// TIA Portal V20 export
FUNCTION_BLOCK "FB_MABS_PNIO"   // FB6, LAD
// stored: Access Published, MemoryReserve 100, Namespace Global, SetENOAutomatically false
   VAR_IN_OUT
      IBP_in : "IB_P01/02/03_in_64bytes_struct";
      IBP_out : "IB_P01/02/03_out_64bytes_struct";
      MABS : "Global.MABS";
   END_VAR
   VAR
      Initializing : Bool;
      Waiting_sw_req : Bool;
      Switching_left : Bool;
      "Switching_left to straight" : Bool;
      "Switching_right to straight" : Bool;
      Switching_right : Bool;
      Switching_done : Bool;
      Tof_life_bit { S7_SetPoint := 'True'} : TON_TIME;
      MABS_sw_timout { S7_SetPoint := 'True'} : TON_TIME;
      "position status_right" : Bool;
      "position status_left" : Bool;
      "position status_straight" : Bool;
      Edge0 : Bool;
      Edge1 : Bool;
      Edge2 : Bool;
      Edge3 : Bool;
      Edge4 : Bool;
      Edge5 : Bool;
      Edge6 : Bool;
      Ton_err_motor_A { S7_SetPoint := 'True'} : TON_TIME;
      Ton_err_motor_B { S7_SetPoint := 'True'} : TON_TIME;
      Ton_err_motor_Com { S7_SetPoint := 'True'} : TON_TIME;
   END_VAR
   VAR_TEMP
      Temp_err_com : Bool;
   END_VAR
   VAR_TEMP   // added for the SCL form of the ladder/FBD networks
      _w1 : Bool;
      _w2 : Bool;
   END_VAR
BEGIN

REGION Network 1: Error motor A & B
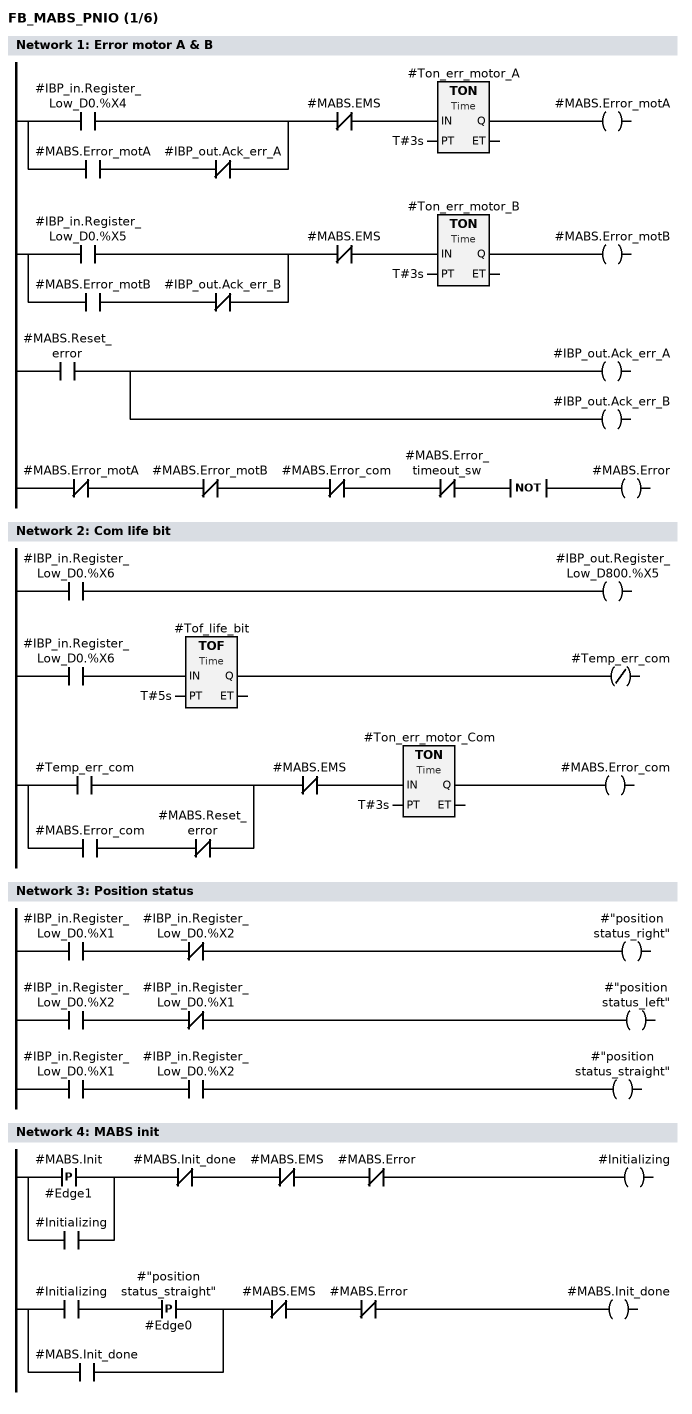
   RUNG wire#powerrail
      Contact( #IBP_in.Register_Low_D0.%X4 )
      wire#w1
      I_Contact( #MABS.EMS )
      { S7_Templates := "time_type := Time" } #Ton_err_motor_A.TON(pt := T#3s, et =>)
      Coil( #MABS.Error_motA )
   END_RUNG
   RUNG wire#powerrail
      Contact( #MABS.Error_motA )
      I_Contact( #IBP_out.Ack_err_A )
   END_RUNG wire#w1
   RUNG wire#powerrail
      Contact( #IBP_in.Register_Low_D0.%X5 )
      wire#w2
      I_Contact( #MABS.EMS )
      { S7_Templates := "time_type := Time" } #Ton_err_motor_B.TON(pt := T#3s, et =>)
      Coil( #MABS.Error_motB )
   END_RUNG
   RUNG wire#powerrail
      Contact( #MABS.Error_motB )
      I_Contact( #IBP_out.Ack_err_B )
   END_RUNG wire#w2
   RUNG wire#powerrail
      Contact( #MABS.Reset_error )
      wire#w3
      Coil( #IBP_out.Ack_err_A )
   END_RUNG
   RUNG wire#w3
      Coil( #IBP_out.Ack_err_B )
   END_RUNG
   RUNG wire#powerrail
      I_Contact( #MABS.Error_motA )
      I_Contact( #MABS.Error_motB )
      I_Contact( #MABS.Error_com )
      I_Contact( #MABS.Error_timeout_sw )
      Not()
      Coil( #MABS.Error )
   END_RUNG
   // the same network as SCL:
   #Ton_err_motor_A(IN := (#IBP_in.Register_Low_D0.%X4 OR (#MABS.Error_motA AND NOT #IBP_out.Ack_err_A)) AND NOT #MABS.EMS,   // TON
                    PT := T#3s);
   #MABS.Error_motA := #Ton_err_motor_A.Q;
   #Ton_err_motor_B(IN := (#IBP_in.Register_Low_D0.%X5 OR (#MABS.Error_motB AND NOT #IBP_out.Ack_err_B)) AND NOT #MABS.EMS,   // TON
                    PT := T#3s);
   #MABS.Error_motB := #Ton_err_motor_B.Q;
   #IBP_out.Ack_err_A := #MABS.Reset_error;
   #IBP_out.Ack_err_B := #MABS.Reset_error;
   #MABS.Error := NOT (NOT #MABS.Error_motA AND NOT #MABS.Error_motB AND NOT #MABS.Error_com AND NOT #MABS.Error_timeout_sw);
END_REGION

REGION Network 2: Com life bit
   RUNG wire#powerrail
      Contact( #IBP_in.Register_Low_D0.%X6 )
      Coil( #IBP_out.Register_Low_D800.%X5 )
   END_RUNG
   RUNG wire#powerrail
      Contact( #IBP_in.Register_Low_D0.%X6 )
      { S7_Templates := "time_type := Time" } #Tof_life_bit.TOF(pt := T#5s, et =>)
      I_Coil( #Temp_err_com )
   END_RUNG
   RUNG wire#powerrail
      Contact( #Temp_err_com )
      wire#w1
      I_Contact( #MABS.EMS )
      { S7_Templates := "time_type := Time" } #Ton_err_motor_Com.TON(pt := T#3s, et =>)
      Coil( #MABS.Error_com )
   END_RUNG
   RUNG wire#powerrail
      Contact( #MABS.Error_com )
      I_Contact( #MABS.Reset_error )
   END_RUNG wire#w1
   // the same network as SCL:
   #IBP_out.Register_Low_D800.%X5 := #IBP_in.Register_Low_D0.%X6;
   #Tof_life_bit(IN := #IBP_in.Register_Low_D0.%X6, PT := T#5s);   // TOF
   #Temp_err_com := NOT #Tof_life_bit.Q;
   #Ton_err_motor_Com(IN := (#Temp_err_com OR (#MABS.Error_com AND NOT #MABS.Reset_error)) AND NOT #MABS.EMS,   // TON
                      PT := T#3s);
   #MABS.Error_com := #Ton_err_motor_Com.Q;
END_REGION

REGION Network 3: Position status
   RUNG wire#powerrail
      Contact( #IBP_in.Register_Low_D0.%X1 )
      I_Contact( #IBP_in.Register_Low_D0.%X2 )
      Coil( #"position status_right" )
   END_RUNG
   RUNG wire#powerrail
      Contact( #IBP_in.Register_Low_D0.%X2 )
      I_Contact( #IBP_in.Register_Low_D0.%X1 )
      Coil( #"position status_left" )
   END_RUNG
   RUNG wire#powerrail
      Contact( #IBP_in.Register_Low_D0.%X1 )
      Contact( #IBP_in.Register_Low_D0.%X2 )
      Coil( #"position status_straight" )
   END_RUNG
   // the same network as SCL:
   #"position status_right" := #IBP_in.Register_Low_D0.%X1 AND NOT #IBP_in.Register_Low_D0.%X2;
   #"position status_left" := #IBP_in.Register_Low_D0.%X2 AND NOT #IBP_in.Register_Low_D0.%X1;
   #"position status_straight" := #IBP_in.Register_Low_D0.%X1 AND #IBP_in.Register_Low_D0.%X2;
END_REGION

REGION Network 4: MABS init
   RUNG wire#powerrail
      P_Contact(operand := #MABS.Init, bit := #Edge1)
      wire#w1
      I_Contact( #MABS.Init_done )
      I_Contact( #MABS.EMS )
      I_Contact( #MABS.Error )
      Coil( #Initializing )
   END_RUNG
   RUNG wire#powerrail
      Contact( #Initializing )
   END_RUNG wire#w1
   RUNG wire#powerrail
      Contact( #Initializing )
      P_Contact(operand := #"position status_straight", bit := #Edge0)
      wire#w2
      I_Contact( #MABS.EMS )
      I_Contact( #MABS.Error )
      Coil( #MABS.Init_done )
   END_RUNG
   RUNG wire#powerrail
      Contact( #MABS.Init_done )
   END_RUNG wire#w2
   // the same network as SCL:
   #_w1 := #MABS.Init AND NOT #Edge1;   // rising edge of #MABS.Init
   #Edge1 := #MABS.Init;
   #Initializing := (#_w1 OR #Initializing) AND NOT #MABS.Init_done AND NOT #MABS.EMS AND NOT #MABS.Error;
   #_w2 := #Initializing AND #"position status_straight" AND NOT #Edge0;   // rising edge of #"position status_straight"
   #Edge0 := #"position status_straight";
   #MABS.Init_done := (#_w2 OR #MABS.Init_done) AND NOT #MABS.EMS AND NOT #MABS.Error;
END_REGION

REGION Network 5: MABS ready
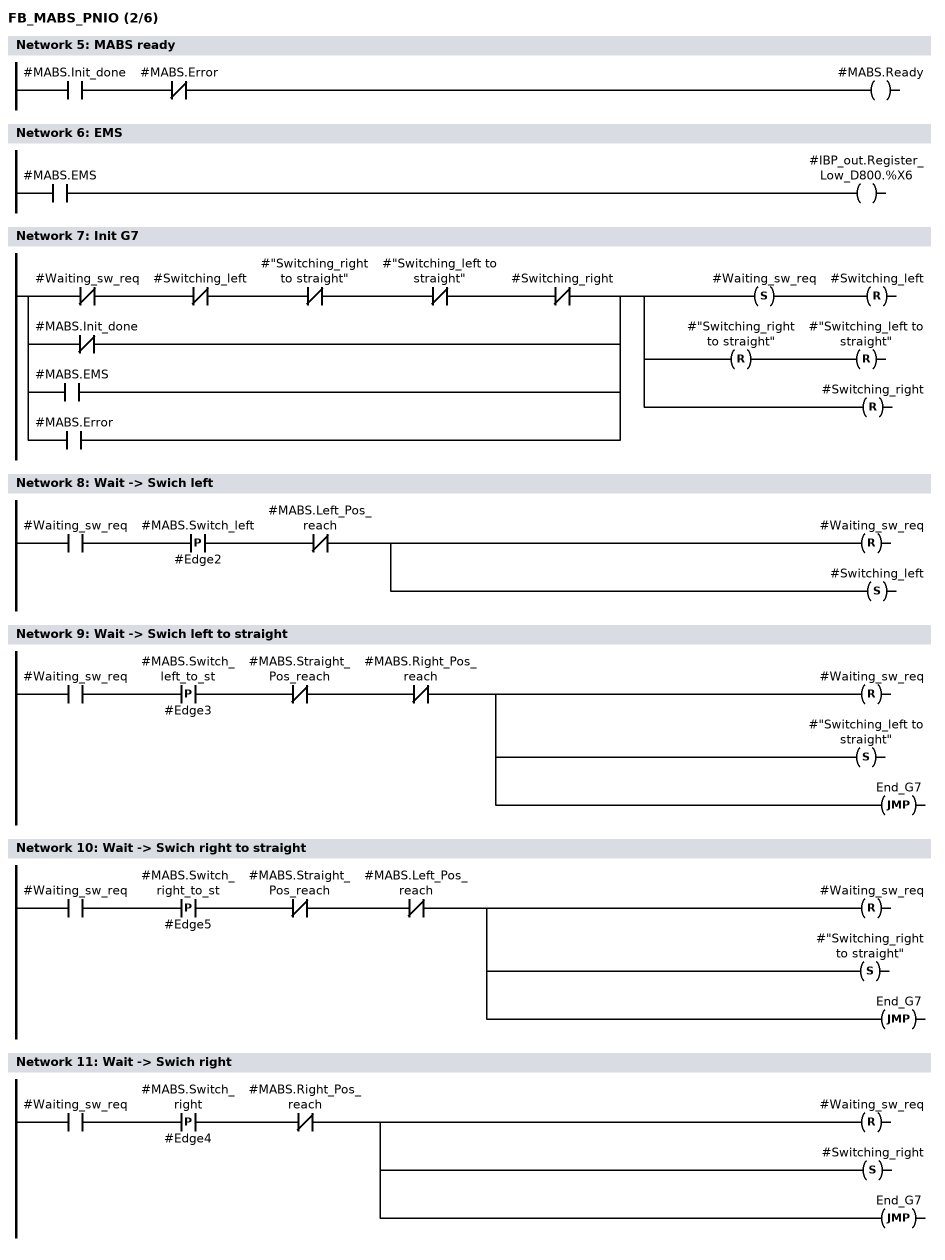
   RUNG wire#powerrail
      Contact( #MABS.Init_done )
      I_Contact( #MABS.Error )
      Coil( #MABS.Ready )
   END_RUNG
   // the same network as SCL:
   #MABS.Ready := #MABS.Init_done AND NOT #MABS.Error;
END_REGION

REGION Network 6: EMS
   RUNG wire#powerrail
      Contact( #MABS.EMS )
      Coil( #IBP_out.Register_Low_D800.%X6 )
   END_RUNG
   // the same network as SCL:
   #IBP_out.Register_Low_D800.%X6 := #MABS.EMS;
END_REGION

REGION Network 7: Init G7
   RUNG wire#powerrail
      I_Contact( #Waiting_sw_req )
      I_Contact( #Switching_left )
      I_Contact( #"Switching_right to straight" )
      I_Contact( #"Switching_left to straight" )
      I_Contact( #Switching_right )
      wire#w1
      S_Coil( #Waiting_sw_req )
      R_Coil( #Switching_left )
   END_RUNG
   RUNG wire#powerrail
      I_Contact( #MABS.Init_done )
   END_RUNG wire#w1
   RUNG wire#powerrail
      Contact( #MABS.EMS )
   END_RUNG wire#w1
   RUNG wire#powerrail
      Contact( #MABS.Error )
   END_RUNG wire#w1
   RUNG wire#w1
      R_Coil( #"Switching_right to straight" )
      R_Coil( #"Switching_left to straight" )
   END_RUNG
   RUNG wire#w1
      R_Coil( #Switching_right )
   END_RUNG
   // the same network as SCL:
   #_w1 := (NOT #Waiting_sw_req AND NOT #Switching_left AND NOT #"Switching_right to straight" AND NOT #"Switching_left to straight" AND NOT #Switching_right) OR NOT #MABS.Init_done OR #MABS.EMS OR #MABS.Error;
   IF #_w1 THEN
       #Waiting_sw_req := TRUE;
       #Switching_left := FALSE;
       #"Switching_right to straight" := FALSE;
       #"Switching_left to straight" := FALSE;
       #Switching_right := FALSE;
   END_IF;
END_REGION

REGION Network 8: Wait -> Swich left
   RUNG wire#powerrail
      Contact( #Waiting_sw_req )
      P_Contact(operand := #MABS.Switch_left, bit := #Edge2)
      I_Contact( #MABS.Left_Pos_reach )
      wire#w1
      R_Coil( #Waiting_sw_req )
   END_RUNG
   RUNG wire#w1
      S_Coil( #Switching_left )
   END_RUNG
   // the same network as SCL:
   #_w1 := #Waiting_sw_req AND #MABS.Switch_left AND NOT #Edge2;   // rising edge of #MABS.Switch_left
   #Edge2 := #MABS.Switch_left;
   IF #_w1 AND NOT #MABS.Left_Pos_reach THEN
       #Waiting_sw_req := FALSE;
       #Switching_left := TRUE;
   END_IF;
END_REGION

REGION Network 9: Wait -> Swich left to straight
   RUNG wire#powerrail
      Contact( #Waiting_sw_req )
      P_Contact(operand := #MABS.Switch_left_to_st, bit := #Edge3)
      I_Contact( #MABS.Straight_Pos_reach )
      I_Contact( #MABS.Right_Pos_reach )
      wire#w1
      R_Coil( #Waiting_sw_req )
   END_RUNG
   RUNG wire#w1
      S_Coil( #"Switching_left to straight" )
   END_RUNG
   RUNG wire#w1
      JumpCoil( End_G7 )
   END_RUNG
   // the same network as SCL:
   #_w1 := #Waiting_sw_req AND #MABS.Switch_left_to_st AND NOT #Edge3;   // rising edge of #MABS.Switch_left_to_st
   #Edge3 := #MABS.Switch_left_to_st;
   #_w2 := #_w1 AND NOT #MABS.Straight_Pos_reach AND NOT #MABS.Right_Pos_reach;
   IF #_w2 THEN
       #Waiting_sw_req := FALSE;
       #"Switching_left to straight" := TRUE;
       GOTO End_G7;
   END_IF;
END_REGION

REGION Network 10: Wait -> Swich right to straight
   RUNG wire#powerrail
      Contact( #Waiting_sw_req )
      P_Contact(operand := #MABS.Switch_right_to_st, bit := #Edge5)
      I_Contact( #MABS.Straight_Pos_reach )
      I_Contact( #MABS.Left_Pos_reach )
      wire#w1
      R_Coil( #Waiting_sw_req )
   END_RUNG
   RUNG wire#w1
      S_Coil( #"Switching_right to straight" )
   END_RUNG
   RUNG wire#w1
      JumpCoil( End_G7 )
   END_RUNG
   // the same network as SCL:
   #_w1 := #Waiting_sw_req AND #MABS.Switch_right_to_st AND NOT #Edge5;   // rising edge of #MABS.Switch_right_to_st
   #Edge5 := #MABS.Switch_right_to_st;
   #_w2 := #_w1 AND NOT #MABS.Straight_Pos_reach AND NOT #MABS.Left_Pos_reach;
   IF #_w2 THEN
       #Waiting_sw_req := FALSE;
       #"Switching_right to straight" := TRUE;
       GOTO End_G7;
   END_IF;
END_REGION

REGION Network 11: Wait -> Swich right
   RUNG wire#powerrail
      Contact( #Waiting_sw_req )
      P_Contact(operand := #MABS.Switch_right, bit := #Edge4)
      I_Contact( #MABS.Right_Pos_reach )
      wire#w1
      R_Coil( #Waiting_sw_req )
   END_RUNG
   RUNG wire#w1
      S_Coil( #Switching_right )
   END_RUNG
   RUNG wire#w1
      JumpCoil( End_G7 )
   END_RUNG
   // the same network as SCL:
   #_w1 := #Waiting_sw_req AND #MABS.Switch_right AND NOT #Edge4;   // rising edge of #MABS.Switch_right
   #Edge4 := #MABS.Switch_right;
   #_w2 := #_w1 AND NOT #MABS.Right_Pos_reach;
   IF #_w2 THEN
       #Waiting_sw_req := FALSE;
       #Switching_right := TRUE;
       GOTO End_G7;
   END_IF;
END_REGION

REGION Network 12: Swich right -> Wait
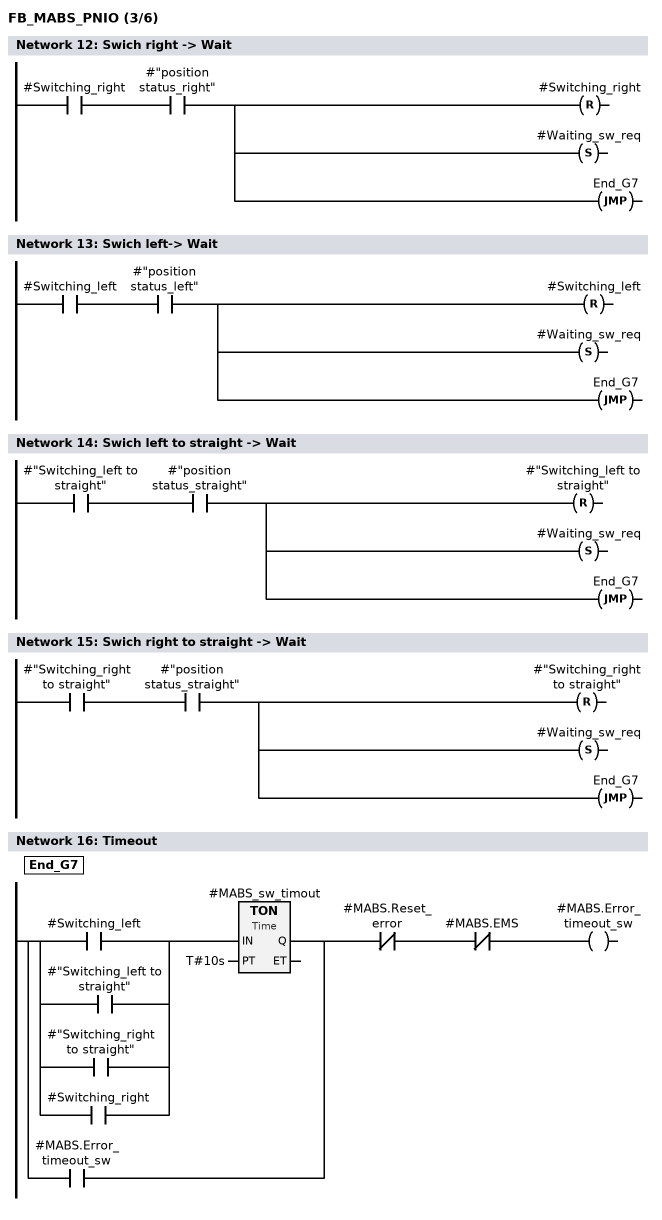
   RUNG wire#powerrail
      Contact( #Switching_right )
      Contact( #"position status_right" )
      wire#w1
      R_Coil( #Switching_right )
   END_RUNG
   RUNG wire#w1
      S_Coil( #Waiting_sw_req )
   END_RUNG
   RUNG wire#w1
      JumpCoil( End_G7 )
   END_RUNG
   // the same network as SCL:
   #_w1 := #Switching_right AND #"position status_right";
   IF #_w1 THEN
       #Switching_right := FALSE;
       #Waiting_sw_req := TRUE;
       GOTO End_G7;
   END_IF;
END_REGION

REGION Network 13: Swich left-> Wait
   RUNG wire#powerrail
      Contact( #Switching_left )
      Contact( #"position status_left" )
      wire#w1
      R_Coil( #Switching_left )
   END_RUNG
   RUNG wire#w1
      S_Coil( #Waiting_sw_req )
   END_RUNG
   RUNG wire#w1
      JumpCoil( End_G7 )
   END_RUNG
   // the same network as SCL:
   #_w1 := #Switching_left AND #"position status_left";
   IF #_w1 THEN
       #Switching_left := FALSE;
       #Waiting_sw_req := TRUE;
       GOTO End_G7;
   END_IF;
END_REGION

REGION Network 14: Swich left to straight -> Wait
   RUNG wire#powerrail
      Contact( #"Switching_left to straight" )
      Contact( #"position status_straight" )
      wire#w1
      R_Coil( #"Switching_left to straight" )
   END_RUNG
   RUNG wire#w1
      S_Coil( #Waiting_sw_req )
   END_RUNG
   RUNG wire#w1
      JumpCoil( End_G7 )
   END_RUNG
   // the same network as SCL:
   #_w1 := #"Switching_left to straight" AND #"position status_straight";
   IF #_w1 THEN
       #"Switching_left to straight" := FALSE;
       #Waiting_sw_req := TRUE;
       GOTO End_G7;
   END_IF;
END_REGION

REGION Network 15: Swich right to straight -> Wait
   RUNG wire#powerrail
      Contact( #"Switching_right to straight" )
      Contact( #"position status_straight" )
      wire#w1
      R_Coil( #"Switching_right to straight" )
   END_RUNG
   RUNG wire#w1
      S_Coil( #Waiting_sw_req )
   END_RUNG
   RUNG wire#w1
      JumpCoil( End_G7 )
   END_RUNG
   // the same network as SCL:
   #_w1 := #"Switching_right to straight" AND #"position status_straight";
   IF #_w1 THEN
       #"Switching_right to straight" := FALSE;
       #Waiting_sw_req := TRUE;
       GOTO End_G7;
   END_IF;
END_REGION

REGION Network 16: Timeout
   Label( End_G7 )
   RUNG wire#powerrail
      Contact( #Switching_left )
      wire#w1
      { S7_Templates := "time_type := Time" } #MABS_sw_timout.TON(pt := T#10s, et =>)
      wire#w2
      I_Contact( #MABS.Reset_error )
      I_Contact( #MABS.EMS )
      Coil( #MABS.Error_timeout_sw )
   END_RUNG
   RUNG wire#powerrail
      Contact( #"Switching_left to straight" )
   END_RUNG wire#w1
   RUNG wire#powerrail
      Contact( #"Switching_right to straight" )
   END_RUNG wire#w1
   RUNG wire#powerrail
      Contact( #Switching_right )
   END_RUNG wire#w1
   RUNG wire#powerrail
      Contact( #MABS.Error_timeout_sw )
   END_RUNG wire#w2
   // the same network as SCL:
   End_G7:
   #MABS_sw_timout(IN := #Switching_left OR #"Switching_left to straight" OR #"Switching_right to straight" OR #Switching_right,   // TON
                   PT := T#10s);
   #MABS.Error_timeout_sw := (#MABS_sw_timout.Q OR #MABS.Error_timeout_sw) AND NOT #MABS.Reset_error AND NOT #MABS.EMS;
END_REGION

REGION Network 17: Postion reached + origin sensor
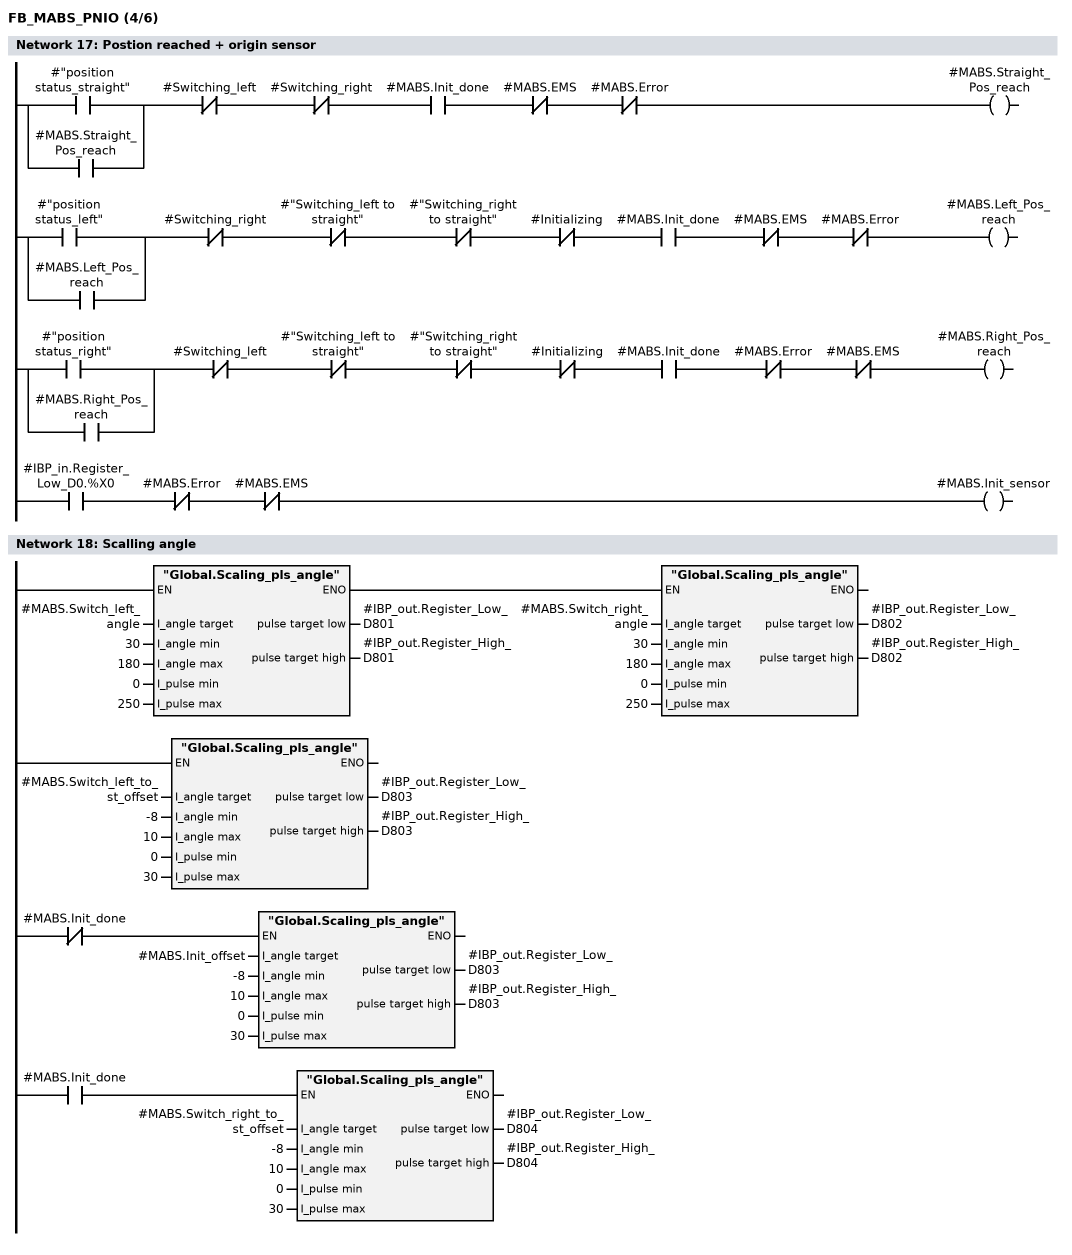
   RUNG wire#powerrail
      Contact( #"position status_straight" )
      wire#w1
      I_Contact( #Switching_left )
      I_Contact( #Switching_right )
      Contact( #MABS.Init_done )
      I_Contact( #MABS.EMS )
      I_Contact( #MABS.Error )
      Coil( #MABS.Straight_Pos_reach )
   END_RUNG
   RUNG wire#powerrail
      Contact( #MABS.Straight_Pos_reach )
   END_RUNG wire#w1
   RUNG wire#powerrail
      Contact( #"position status_left" )
      wire#w2
      I_Contact( #Switching_right )
      I_Contact( #"Switching_left to straight" )
      I_Contact( #"Switching_right to straight" )
      I_Contact( #Initializing )
      Contact( #MABS.Init_done )
      I_Contact( #MABS.EMS )
      I_Contact( #MABS.Error )
      Coil( #MABS.Left_Pos_reach )
   END_RUNG
   RUNG wire#powerrail
      Contact( #MABS.Left_Pos_reach )
   END_RUNG wire#w2
   RUNG wire#powerrail
      Contact( #"position status_right" )
      wire#w3
      I_Contact( #Switching_left )
      I_Contact( #"Switching_left to straight" )
      I_Contact( #"Switching_right to straight" )
      I_Contact( #Initializing )
      Contact( #MABS.Init_done )
      I_Contact( #MABS.Error )
      I_Contact( #MABS.EMS )
      Coil( #MABS.Right_Pos_reach )
   END_RUNG
   RUNG wire#powerrail
      Contact( #MABS.Right_Pos_reach )
   END_RUNG wire#w3
   RUNG wire#powerrail
      Contact( #IBP_in.Register_Low_D0.%X0 )
      I_Contact( #MABS.Error )
      I_Contact( #MABS.EMS )
      Coil( #MABS.Init_sensor )
   END_RUNG
   // the same network as SCL:
   #MABS.Straight_Pos_reach := (#"position status_straight" OR #MABS.Straight_Pos_reach) AND NOT #Switching_left AND NOT #Switching_right AND #MABS.Init_done AND NOT #MABS.EMS AND NOT #MABS.Error;
   #MABS.Left_Pos_reach := (#"position status_left" OR #MABS.Left_Pos_reach) AND NOT #Switching_right AND NOT #"Switching_left to straight" AND NOT #"Switching_right to straight" AND NOT #Initializing AND #MABS.Init_done AND NOT #MABS.EMS AND NOT #MABS.Error;
   #MABS.Right_Pos_reach := (#"position status_right" OR #MABS.Right_Pos_reach) AND NOT #Switching_left AND NOT #"Switching_left to straight" AND NOT #"Switching_right to straight" AND NOT #Initializing AND #MABS.Init_done AND NOT #MABS.Error AND NOT #MABS.EMS;
   #MABS.Init_sensor := #IBP_in.Register_Low_D0.%X0 AND NOT #MABS.Error AND NOT #MABS.EMS;
END_REGION

REGION Network 18: Scalling angle
   RUNG wire#powerrail
      "Global.Scaling_pls_angle"("I_angle target" := #MABS.Switch_left_angle, "I_angle min" := 30, "I_angle max" := 180, "I_pulse min" := 0, "I_pulse max" := 250, "pulse target low" => #IBP_out.Register_Low_D801, "pulse target high" => #IBP_out.Register_High_D801)
      "Global.Scaling_pls_angle"("I_angle target" := #MABS.Switch_right_angle, "I_angle min" := 30, "I_angle max" := 180, "I_pulse min" := 0, "I_pulse max" := 250, "pulse target low" => #IBP_out.Register_Low_D802, "pulse target high" => #IBP_out.Register_High_D802)
   END_RUNG
   RUNG wire#powerrail
      "Global.Scaling_pls_angle"("I_angle target" := #MABS.Switch_left_to_st_offset, "I_angle min" := -8, "I_angle max" := 10, "I_pulse min" := 0, "I_pulse max" := 30, "pulse target low" => #IBP_out.Register_Low_D803, "pulse target high" => #IBP_out.Register_High_D803)
   END_RUNG
   RUNG wire#powerrail
      I_Contact( #MABS.Init_done )
      "Global.Scaling_pls_angle"("I_angle target" := #MABS.Init_offset, "I_angle min" := -8, "I_angle max" := 10, "I_pulse min" := 0, "I_pulse max" := 30, "pulse target low" => #IBP_out.Register_Low_D803, "pulse target high" => #IBP_out.Register_High_D803)
   END_RUNG
   RUNG wire#powerrail
      Contact( #MABS.Init_done )
      "Global.Scaling_pls_angle"("I_angle target" := #MABS.Switch_right_to_st_offset, "I_angle min" := -8, "I_angle max" := 10, "I_pulse min" := 0, "I_pulse max" := 30, "pulse target low" => #IBP_out.Register_Low_D804, "pulse target high" => #IBP_out.Register_High_D804)
   END_RUNG
   // the same network as SCL:
   "Global.Scaling_pls_angle"("I_angle target" := #MABS.Switch_left_angle,
                           "I_angle min" := 30,
                           "I_angle max" := 180,
                           "I_pulse min" := 0,
                           "I_pulse max" := 250,
                           "pulse target low" => #IBP_out.Register_Low_D801,
                           "pulse target high" => #IBP_out.Register_High_D801,
                           ENO => #_w1);
   IF #_w1 THEN
       "Global.Scaling_pls_angle"("I_angle target" := #MABS.Switch_right_angle,
                               "I_angle min" := 30,
                               "I_angle max" := 180,
                               "I_pulse min" := 0,
                               "I_pulse max" := 250,
                               "pulse target low" => #IBP_out.Register_Low_D802,
                               "pulse target high" => #IBP_out.Register_High_D802);
   END_IF;
   "Global.Scaling_pls_angle"("I_angle target" := #MABS.Switch_left_to_st_offset,
                           "I_angle min" := -8,
                           "I_angle max" := 10,
                           "I_pulse min" := 0,
                           "I_pulse max" := 30,
                           "pulse target low" => #IBP_out.Register_Low_D803,
                           "pulse target high" => #IBP_out.Register_High_D803);
   IF NOT #MABS.Init_done THEN
       "Global.Scaling_pls_angle"("I_angle target" := #MABS.Init_offset,
                               "I_angle min" := -8,
                               "I_angle max" := 10,
                               "I_pulse min" := 0,
                               "I_pulse max" := 30,
                               "pulse target low" => #IBP_out.Register_Low_D803,
                               "pulse target high" => #IBP_out.Register_High_D803);
   END_IF;
   IF #MABS.Init_done THEN
       "Global.Scaling_pls_angle"("I_angle target" := #MABS.Switch_right_to_st_offset,
                               "I_angle min" := -8,
                               "I_angle max" := 10,
                               "I_pulse min" := 0,
                               "I_pulse max" := 30,
                               "pulse target low" => #IBP_out.Register_Low_D804,
                               "pulse target high" => #IBP_out.Register_High_D804);
   END_IF;
END_REGION

REGION Network 19: Swing direction
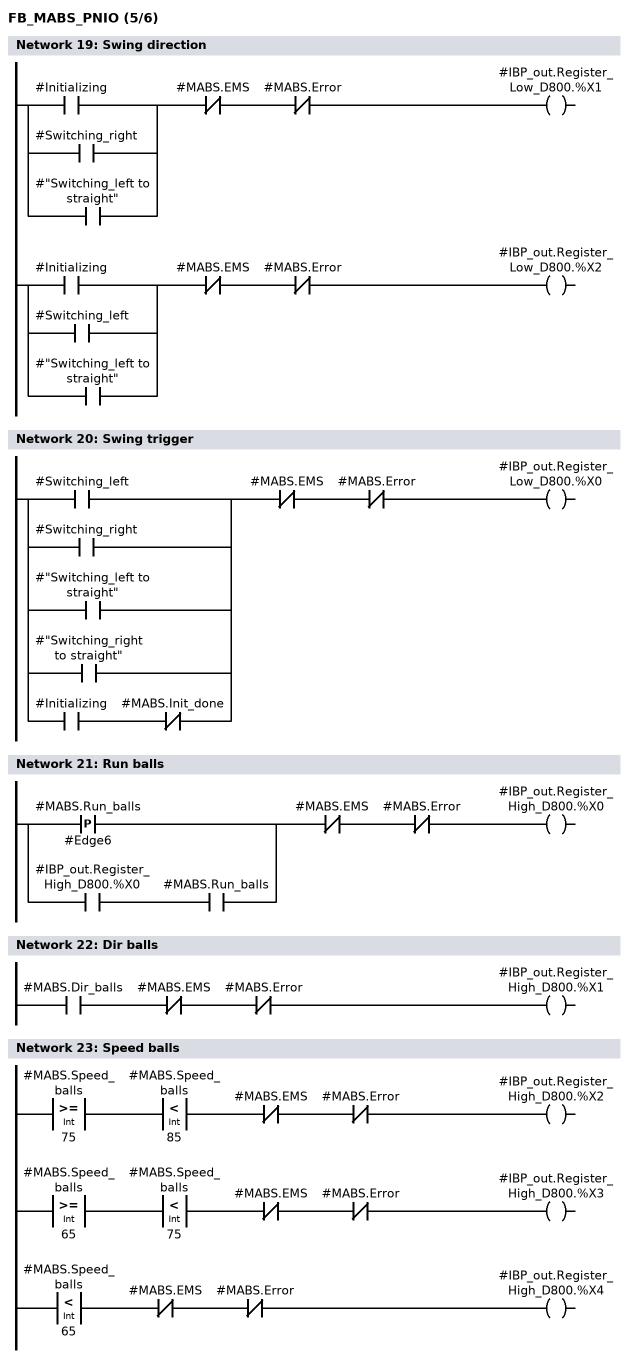
   RUNG wire#powerrail
      Contact( #Initializing )
      wire#w1
      I_Contact( #MABS.EMS )
      I_Contact( #MABS.Error )
      Coil( #IBP_out.Register_Low_D800.%X1 )
   END_RUNG
   RUNG wire#powerrail
      Contact( #Switching_right )
   END_RUNG wire#w1
   RUNG wire#powerrail
      Contact( #"Switching_left to straight" )
   END_RUNG wire#w1
   RUNG wire#powerrail
      Contact( #Initializing )
      wire#w2
      I_Contact( #MABS.EMS )
      I_Contact( #MABS.Error )
      Coil( #IBP_out.Register_Low_D800.%X2 )
   END_RUNG
   RUNG wire#powerrail
      Contact( #Switching_left )
   END_RUNG wire#w2
   RUNG wire#powerrail
      Contact( #"Switching_left to straight" )
   END_RUNG wire#w2
   // the same network as SCL:
   #IBP_out.Register_Low_D800.%X1 := (#Initializing OR #Switching_right OR #"Switching_left to straight") AND NOT #MABS.EMS AND NOT #MABS.Error;
   #IBP_out.Register_Low_D800.%X2 := (#Initializing OR #Switching_left OR #"Switching_left to straight") AND NOT #MABS.EMS AND NOT #MABS.Error;
END_REGION

REGION Network 20: Swing trigger
   RUNG wire#powerrail
      Contact( #Switching_left )
      wire#w1
      I_Contact( #MABS.EMS )
      I_Contact( #MABS.Error )
      Coil( #IBP_out.Register_Low_D800.%X0 )
   END_RUNG
   RUNG wire#powerrail
      Contact( #Switching_right )
   END_RUNG wire#w1
   RUNG wire#powerrail
      Contact( #"Switching_left to straight" )
   END_RUNG wire#w1
   RUNG wire#powerrail
      Contact( #"Switching_right to straight" )
   END_RUNG wire#w1
   RUNG wire#powerrail
      Contact( #Initializing )
      I_Contact( #MABS.Init_done )
   END_RUNG wire#w1
   // the same network as SCL:
   #IBP_out.Register_Low_D800.%X0 := (#Switching_left OR #Switching_right OR #"Switching_left to straight" OR #"Switching_right to straight" OR (#Initializing AND NOT #MABS.Init_done)) AND NOT #MABS.EMS AND NOT #MABS.Error;
END_REGION

REGION Network 21: Run balls
   RUNG wire#powerrail
      P_Contact(operand := #MABS.Run_balls, bit := #Edge6)
      wire#w1
      I_Contact( #MABS.EMS )
      I_Contact( #MABS.Error )
      Coil( #IBP_out.Register_High_D800.%X0 )
   END_RUNG
   RUNG wire#powerrail
      Contact( #IBP_out.Register_High_D800.%X0 )
      Contact( #MABS.Run_balls )
   END_RUNG wire#w1
   // the same network as SCL:
   #_w1 := #MABS.Run_balls AND NOT #Edge6;   // rising edge of #MABS.Run_balls
   #Edge6 := #MABS.Run_balls;
   #IBP_out.Register_High_D800.%X0 := (#_w1 OR (#IBP_out.Register_High_D800.%X0 AND #MABS.Run_balls)) AND NOT #MABS.EMS AND NOT #MABS.Error;
END_REGION

REGION Network 22: Dir balls
   RUNG wire#powerrail
      Contact( #MABS.Dir_balls )
      I_Contact( #MABS.EMS )
      I_Contact( #MABS.Error )
      Coil( #IBP_out.Register_High_D800.%X1 )
   END_RUNG
   // the same network as SCL:
   #IBP_out.Register_High_D800.%X1 := #MABS.Dir_balls AND NOT #MABS.EMS AND NOT #MABS.Error;
END_REGION

REGION Network 23: Speed balls
   RUNG wire#powerrail
      { S7_Templates := "SrcType := Int" } GE_Contact(in1 := #MABS.Speed_balls, in2 := 75)
      { S7_Templates := "SrcType := Int" } LT_Contact(in1 := #MABS.Speed_balls, in2 := 85)
      I_Contact( #MABS.EMS )
      I_Contact( #MABS.Error )
      Coil( #IBP_out.Register_High_D800.%X2 )
   END_RUNG
   RUNG wire#powerrail
      { S7_Templates := "SrcType := Int" } GE_Contact(in1 := #MABS.Speed_balls, in2 := 65)
      { S7_Templates := "SrcType := Int" } LT_Contact(in1 := #MABS.Speed_balls, in2 := 75)
      I_Contact( #MABS.EMS )
      I_Contact( #MABS.Error )
      Coil( #IBP_out.Register_High_D800.%X3 )
   END_RUNG
   RUNG wire#powerrail
      { S7_Templates := "SrcType := Int" } LT_Contact(in1 := #MABS.Speed_balls, in2 := 65)
      I_Contact( #MABS.EMS )
      I_Contact( #MABS.Error )
      Coil( #IBP_out.Register_High_D800.%X4 )
   END_RUNG
   // the same network as SCL:
   #IBP_out.Register_High_D800.%X2 := (#MABS.Speed_balls >= 75) AND (#MABS.Speed_balls < 85) AND NOT #MABS.EMS AND NOT #MABS.Error;
   #IBP_out.Register_High_D800.%X3 := (#MABS.Speed_balls >= 65) AND (#MABS.Speed_balls < 75) AND NOT #MABS.EMS AND NOT #MABS.Error;
   #IBP_out.Register_High_D800.%X4 := (#MABS.Speed_balls < 65) AND NOT #MABS.EMS AND NOT #MABS.Error;
END_REGION

REGION Network 24: HMI status
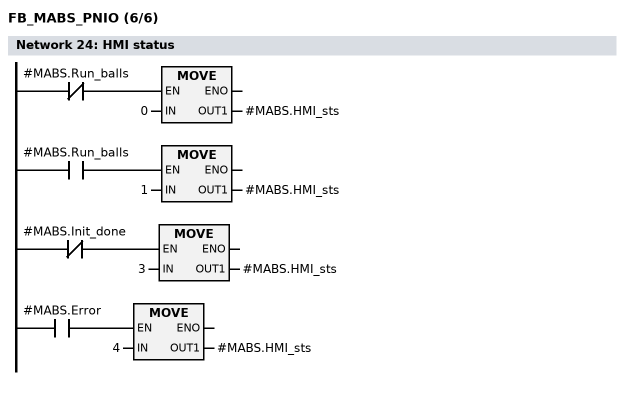
   RUNG wire#powerrail
      I_Contact( #MABS.Run_balls )
      Move(in := 0, out1 => #MABS.HMI_sts)
   END_RUNG
   RUNG wire#powerrail
      Contact( #MABS.Run_balls )
      Move(in := 1, out1 => #MABS.HMI_sts)
   END_RUNG
   RUNG wire#powerrail
      I_Contact( #MABS.Init_done )
      Move(in := 3, out1 => #MABS.HMI_sts)
   END_RUNG
   RUNG wire#powerrail
      Contact( #MABS.Error )
      Move(in := 4, out1 => #MABS.HMI_sts)
   END_RUNG
   // the same network as SCL:
   IF NOT #MABS.Run_balls THEN #MABS.HMI_sts := 0; END_IF;
   IF #MABS.Run_balls THEN #MABS.HMI_sts := 1; END_IF;
   IF NOT #MABS.Init_done THEN #MABS.HMI_sts := 3; END_IF;
   IF #MABS.Error THEN #MABS.HMI_sts := 4; END_IF;
END_REGION
END_FUNCTION_BLOCK
